// TwinCAT 3 PLC project Untitled1
// ProgramVersion: 3.1.4023.0
// libraries:
//   Tc2_SerialCom, * (Beckhoff Automation GmbH)
//   Tc2_Standard, * (Beckhoff Automation GmbH)
//   Tc2_System, * (Beckhoff Automation GmbH)
//   Tc2_Utilities, * (Beckhoff Automation GmbH)
//   Tc3_Database, * (Beckhoff Automation GmbH)
//   Tc3_IotBase, * (Beckhoff Automation GmbH)
//   Tc3_Module, * (Beckhoff Automation GmbH)
// project tree:
//   DUTs/ ST_SelectStructData.TcDUT, ST_SelectStructIMU.TcDUT (not stored)
//   GVLs/ GVL.TcGVL (not stored)
//   / PlcTask_Background.TcTTO (not stored), PlcTask_Buffer.TcTTO (not stored), PlcTask_Send.TcTTO, PlcTask_Read.TcTTO (not stored), PlcTask_Vacuum.TcTTO
//   POUs/ Background_FatigueCam.TcPOU (not stored), Background_GPS.TcPOU, Background_IMU.TcPOU (not stored), Background_Time.TcPOU, Buffer_Data.TcPOU (not stored), Buffer_IMU.TcPOU, FB_FatigueCam_Receive.TcPOU, Get_Data.TcPOU (not stored), Get_IMU.TcPOU, Main_Background.TcPOU (not stored), Main_Read.TcPOU (not stored), Main_Vacuum.TcPOU, Read_IMU.TcPOU (not stored), Read_Pressure.TcPOU, Read_Payload.TcPOU, Main_Buffer.TcPOU (not stored), Main_Send.TcPOU, Read_FatigueCam.TcPOU (not stored), Read_GPS.TcPOU, Read_ID.TcPOU, Save_Data.TcPOU (not stored), Save_IMU.TcPOU (not stored), Send.TcPOU, Send_IMU.TcPOU, Vacuum_Buffer_Data.TcPOU, Vacuum_Buffer_Data_2.TcPOU, Vacuum_Buffer_IMU.TcPOU, Vacuum_Buffer_IMU_2.TcPOU, Vacuum_Data.TcPOU (not stored), Vacuum_IMU.TcPOU (not stored)

CONFIGURATION Untitled1
    RESOURCE PLC ON TwinCAT3
        TASK PlcTask_Send(INTERVAL := T#4332.9us, PRIORITY := 21);
        TASK PlcTask_Vacuum(INTERVAL := T#333.3us, PRIORITY := 16);
        PROGRAM Main_Send WITH PlcTask_Send : Main_Send;
        PROGRAM Main_Vacuum WITH PlcTask_Vacuum : Main_Vacuum;
    END_RESOURCE
END_CONFIGURATION

// ---- DUTs/ST_SelectStructData.TcDUT
TYPE ST_SelectStructData :
STRUCT
	datetime: STRING(255);
	trailer_id_lead: LINT;
	trailer_id_rear: LINT;
	latitude: REAL;
	longitude: REAL;
	speed: REAL;
	overspeed: LINT;
	payload_lead: REAL;
	payload_rear: REAL;
	overload_lead: LINT;
	overload_rear: LINT;
	pressure_lead: REAL;
	pressure_rear: REAL;
	overpressure_lead: LINT;
	overpressure_rear: LINT;
	event_code: LINT;
END_STRUCT
END_TYPE

// ---- POUs/Main_Send.TcPOU
PROGRAM Main_Send
VAR	
	Done		: BOOL;
	New_Data	: BOOL;
	New_IMU		: BOOL;
	Sent		: BOOL;
	Saved		: BOOL;
	Sent_Data	: BOOL;
	Sent_IMU	: BOOL;
	Saved_Data	: BOOL;
	Saved_IMU	: BOOL;
	
	nState		: INT;

END_VAR

(* get data from database *)
Get_Data();
Get_IMU();

New_Data := Get_Data.Done;
New_IMU := Get_IMU.Done;
 
IF New_Data AND New_IMU THEN
	IF NOT Sent THEN
		(* send data to aws iot core *)
		Send();
		
		IF Send.Published_Data AND Send.Published_IMU THEN
			Sent	:= TRUE;
		END_IF	
		
	ELSE
		IF Save_Data.Done AND Save_IMU.Done THEN
			Saved := TRUE;
		END_IF	
		
	END_IF
	
ELSE
	Sent	:= FALSE;
	Saved 	:= FALSE;
	
END_IF

Save_Data();	
Save_IMU();

END_PROGRAM

// ---- POUs/Get_IMU.TcPOU
PROGRAM Get_IMU
VAR
	fbSqlDatabase	: FB_SQLDatabaseEvt(sNetID := '', tTimeout := T#1000S);
	fbSqlCommand	: FB_SQLCommandEvt(sNetID := '', tTimeout := T#1000S);
	fbSqlCommand2	: FB_SQLCommandEvt(sNetID := '', tTimeout := T#1000S);
	fbSqlResult		: FB_SQLResultEvt(sNetID:='', tTimeout   := T#1000S); 
    aReadStruct		: ARRAY[1..2500] OF ST_SelectStructIMU;
	nState			: INT;
	sCmd			: STRING(20000);
	sCmd2			: STRING(20000);
	val1			: INT;
	val2			: INT;
	exec			: BOOL;
	diff			: BOOL;
	rel				: BOOL;
	exec2			: BOOL;
	diff2			: BOOL;	
	rel2			: BOOL;
	exec3			: BOOL;
	diff3			: BOOL;	
	rel3			: BOOL;
	
	count			: ULINT;
	Data_Length		: ULINT;
	datetime		: STRING;
	Done			: BOOL;
	Deleted			: BOOL := TRUE;
	i 				: ULINT;
	
	TimeStr			: ARRAY[1..2500] OF STRING;	
	Trailer_ID_Lead	: ARRAY[1..2500] OF STRING;
	Trailer_ID_Rear	: ARRAY[1..2500] OF STRING;
	Pitch_Lead		: ARRAY[1..2500] OF STRING;
	Roll_Lead		: ARRAY[1..2500] OF STRING;
	AccX_Lead		: ARRAY[1..2500] OF STRING;
	AccY_Lead		: ARRAY[1..2500] OF STRING;
	AccZ_Lead		: ARRAY[1..2500] OF STRING;
	Pitch_Rear		: ARRAY[1..2500] OF STRING;
	Roll_Rear		: ARRAY[1..2500] OF STRING;
	AccX_Rear		: ARRAY[1..2500] OF STRING;
	AccY_Rear		: ARRAY[1..2500] OF STRING;
	AccZ_Rear		: ARRAY[1..2500] OF STRING;
	
	Dbid			: UDINT;
	Switch			: BOOL;
	Pragma_Done		: BOOL;
	bDisconnect		: BOOL;
	
END_VAR

(* get new data only if prev data sent to aws & saved to localdb *)
IF Main_Send.Saved THEN
	Done	:= FALSE;
	Deleted	:= FALSE;
	IF fbSqlDatabase.bConnected THEN
		nState 	:= 1;
	ELSE
		nState 	:= 0;
	END_IF
END_IF

IF Switch THEN
	IF Buffer_IMU.Dbid = Dbid AND Buffer_IMU.fbSqlDatabase.bConnected THEN
		Switch := FALSE;
	END_IF
	
ELSIF Buffer_IMU.Initialized AND Buffer_IMU.fbSqlDatabase.bConnected THEN
	
	CASE nState OF
		
		0:
			//choose db opposite of buffer
			IF Buffer_IMU.Dbid = 2 THEN
				Dbid := 5;
			ELSE
				Dbid := 2;
			END_IF
			
			IF fbSqlDatabase.Connect(Dbid) THEN
				IF fbSqlDatabase.bError THEN
					nState := 255;
				ELSE
					nState := nState + 1;
				END_IF
			END_IF
			
		1:
			IF fbSqlDatabase.CreateCmd(ADR(fbSqlCommand)) THEN
				IF fbSqlDatabase.bError THEN
					nState := 255; 
				ELSE
					nState := nState+1; 
				END_IF
			END_IF
			
		2:	(* execute pragmas *)
			IF NOT Pragma_Done THEN
				sCmd	:= 'PRAGMA journal_mode = WAL; PRAGMA synchronous = NORMAL; PRAGMA temp_store = MEMORY; PRAGMA mmap_size = 30000000000; PRAGMA page_size = 32768; PRAGMA locking_mode = EXCLUSIVE;';
			
				IF fbSQLCommand.Execute(ADR(sCmd), SIZEOF(sCmd)) THEN
					IF fbSQLCommand.bError THEN
						nState := 255; 
					ELSE
						nState 		:= nState+1; 
						Pragma_Done := TRUE;
					END_IF
				END_IF
			
			ELSE
				nState 		:= nState+1;
			END_IF
		
		3:	
			IF Deleted THEN
				nState := nState+1;
			ELSE
				(* delete saved data from buffer *)
				sCmd2	:= 'DELETE FROM buffer_imu WHERE datetime IN (SELECT datetime FROM buffer_imu ORDER BY datetime ASC LIMIT ';
				sCmd2	:= CONCAT(sCmd2, ULINT_TO_STRING(Data_Length));
				sCmd2	:= CONCAT(sCmd2, ');');
				
				IF fbSQLCommand.Execute(ADR(sCmd2), SIZEOF(sCmd2)) THEN
					IF fbSQLCommand.bError THEN
						nState := 255; 
					ELSE
						nState := nState+1; 
						Deleted := TRUE;
					END_IF
				END_IF
			END_IF
			
		4:	
			(* count no of records in buffer *)
			sCmd2 := 'SELECT COUNT(*) FROM `buffer_imu`';
			
			IF fbSQLCommand.ExecuteDataReturn(ADR(sCmd2), SIZEOF(sCmd2), ADR(fbSqlResult)) THEN
				IF fbSQLCommand.bError THEN
					nState := 255; 
				ELSE
					nState := nState+1; 
				END_IF
			END_IF
			
		5:	
			IF fbSqlResult.Read(0, 1, ADR(count), SIZEOF(count), TRUE, TRUE) THEN
				IF fbSqlResult.bError THEN
					nState := 255; 
				ELSE
					nState := nState+1; 
				END_IF
			END_IF
			
		6:
			IF fbSqlResult.Release() THEN
				IF fbSqlResult.bError THEN
					nState := 255;
				ELSE
					nState := nState + 1;
				END_IF
				
			END_IF
			
		7:
			(* determine no of records to select *)
			IF count = 0 THEN
				Data_Length := 0;
				nState := 13;
			
			ELSIF count < 1000 THEN
				Data_Length := count;
				nState := nState+1;
			
			ELSE
				Data_Length := 1000;
				nState := nState+1;
			
			END_IF
			
		8:	
			(* get records from buffer *)
			sCmd2 := 'SELECT * FROM `buffer_imu` ORDER BY datetime ASC LIMIT ';
			sCmd2 := CONCAT(sCmd2, ULINT_TO_STRING(Data_Length));
			
			IF fbSQLCommand.ExecuteDataReturn(ADR(sCmd2), SIZEOF(sCmd2), ADR(fbSqlResult)) THEN
				IF fbSQLCommand.bError THEN
					nState := 255; 
				ELSE
					nState := nState+1; 
				END_IF
			END_IF
			
		9:
			IF fbSqlResult.Read(0, ULINT_TO_UDINT(Data_Length), ADR(aReadStruct), SIZEOF(aReadStruct), TRUE, TRUE) THEN
				IF fbSqlResult.bError THEN
					nState := 255; 
				ELSE
					nState := nState+1; 
				END_IF
			END_IF
			
		10:
			IF fbSqlResult.Release() THEN
				IF fbSqlResult.bError THEN
					nState := 255;
				ELSE
					nState := nState+1;
				END_IF
			END_IF
		
		11:
			(* parse query result *)
			FOR i:=1 TO Data_Length BY 1 DO
				TimeStr[i]			:= aReadStruct[i].datetime;
				
				Trailer_ID_Lead[i]			:= LINT_TO_STRING(aReadStruct[i].trailer_id_lead);
				Trailer_ID_Rear[i]			:= LINT_TO_STRING(aReadStruct[i].trailer_id_rear);
				//RoadSec[i]				:= UINT_TO_STRING(aReadStruct[i].RoadSec);
				Pitch_Lead[i]				:= REAL_TO_STRING(aReadStruct[i].pitch_lead);
				Roll_Lead[i]				:= REAL_TO_STRING(aReadStruct[i].roll_lead);
				AccX_Lead[i]				:= REAL_TO_STRING(aReadStruct[i].ax_lead);
				AccY_Lead[i]				:= REAL_TO_STRING(aReadStruct[i].ay_lead);
				AccZ_Lead[i]				:= REAL_TO_STRING(aReadStruct[i].az_lead);
				Pitch_Rear[i]				:= REAL_TO_STRING(aReadStruct[i].pitch_rear);
				Roll_Rear[i]				:= REAL_TO_STRING(aReadStruct[i].roll_rear);
				AccX_Rear[i]				:= REAL_TO_STRING(aReadStruct[i].ax_rear);
				AccY_Rear[i]				:= REAL_TO_STRING(aReadStruct[i].ay_rear);
				AccZ_Rear[i]				:= REAL_TO_STRING(aReadStruct[i].az_rear);
				
			END_FOR
			
			nState	:= nState + 1;
			
		12:
			Done	:= TRUE;
			
		13:	(* execute pragma optimize *)
			sCmd	:= 'PRAGMA optimize;';
			
			IF fbSQLCommand.Execute(ADR(sCmd), SIZEOF(sCmd)) THEN
				IF fbSQLCommand.bError THEN
					nState := 255; 
				ELSE
					nState := nState+1; 
				END_IF
			END_IF
			
		14:
			//disconnect from db
			IF bDisconnect := fbSqlDatabase.Disconnect() THEN
				IF fbSqlDatabase.bError THEN
					nState := 255;
				ELSE
					nState 		:= 0;
					Switch 		:= TRUE;
					Pragma_Done	:= FALSE;
				END_IF
			END_IF			
		
		255:
			nState	:= 0;	
			
	END_CASE
	
END_IF

END_PROGRAM

// ---- POUs/Buffer_IMU.TcPOU
PROGRAM Buffer_IMU
VAR
	pSec		: WORD;
	diff		: BOOL;
	
	TimeStr		: ARRAY [1..50] OF STRING;
	//Millis		: ARRAY [1..50] OF STRING;
	Trailer_ID_Lead	: ARRAY [1..50] OF STRING;
	//RoadSec		: ARRAY [1..50] OF STRING;
	Pitch_Lead		: ARRAY [1..50] OF STRING;
	Roll_Lead		: ARRAY [1..50] OF STRING;
	AccX_Lead		: ARRAY [1..50] OF STRING;
	AccY_Lead		: ARRAY [1..50] OF STRING;
	AccZ_Lead		: ARRAY [1..50] OF STRING;
	
	Trailer_ID_Rear	: ARRAY [1..50] OF STRING;
	//RoadSec		: ARRAY [1..50] OF STRING;
	Pitch_Rear		: ARRAY [1..50] OF STRING;
	Roll_Rear		: ARRAY [1..50] OF STRING;
	AccX_Rear		: ARRAY [1..50] OF STRING;
	AccY_Rear		: ARRAY [1..50] OF STRING;
	AccZ_Rear		: ARRAY [1..50] OF STRING;
	
	fbSqlDatabase	: FB_SQLDatabaseEvt(sNetID := '', tTimeout := T#1000S);
	fbSqlCommand	: FB_SQLCommandEvt(sNetID := '', tTimeout := T#1000S);
	fbSqlResult		: FB_SQLResultEvt(sNetID:='', tTimeout   := T#1000S); 
	sCmd			: STRING(500000);
	sCmd2			: STRING(500000);
	nState			: INT;
	nState_Switch	: INT;
	
	aReadStruct		: ST_SelectStructIMU;
	aReadStruct_2	: ST_SelectStructIMU;
	Timestamp		: DT;
	Timestamp_2		: DT; 
	
	Initialized		: BOOL := FALSE;
	Done			: BOOL;
	i				: INT;
	Pragma_Done		: BOOL;
	Counter			: ULINT;
	
	Dbid			: UDINT;
	
	bDisconnect		: BOOL;
END_VAR

(* convert to strings *)
//PrimeMover_ID		:= Read_ID.PrimeMover_ID;
TimeStr				:= Read_IMU.TimeStr;
//Millis			:= Read_IMU.Millis;
Trailer_ID_Lead		:= Read_IMU.Trailer_ID_Lead;
Pitch_Lead			:= Read_IMU.Pitch_Lead;
Roll_Lead			:= Read_IMU.Roll_Lead;
AccX_Lead			:= Read_IMU.AccX_Lead;
AccY_Lead			:= Read_IMU.AccY_Lead;
AccZ_Lead			:= Read_IMU.AccZ_Lead;

Trailer_ID_Rear		:= Read_IMU.Trailer_ID_Rear;
Pitch_Rear			:= Read_IMU.Pitch_Rear;
Roll_Rear			:= Read_IMU.Roll_Rear;
AccX_Rear			:= Read_IMU.AccX_Rear;
AccY_Rear			:= Read_IMU.AccY_Rear;
AccZ_Rear			:= Read_IMU.AccZ_Rear;

IF NOT Initialized THEN
	
	//initialization (choose which database for buffer)
	CASE nState OF
				
		0:
			(* connect to buffer_imu *)	
			IF Vacuum_Buffer_IMU.Vacuumed THEN
				
				Dbid := 2;		
				IF fbSqlDatabase.Connect(Dbid) THEN
					IF fbSqlDatabase.bError THEN
						nState := 255; 
					ELSE
						nState := nState+1;
					END_IF
				END_IF
				
			END_IF
			
			
		1:
			IF fbSqlDatabase.CreateCmd(ADR(fbSqlCommand)) THEN
				IF fbSqlDatabase.bError THEN
					nState := 255; 
				ELSE
					nState := nState+1; 
				END_IF
			END_IF
			
		2:	(* execute pragmas *)
			sCmd	:= 'PRAGMA journal_mode = WAL; PRAGMA synchronous = NORMAL; PRAGMA temp_store = MEMORY; PRAGMA mmap_size = 30000000000; PRAGMA page_size = 32768; PRAGMA locking_mode = EXCLUSIVE;';
			
			IF fbSQLCommand.Execute(ADR(sCmd), SIZEOF(sCmd)) THEN
				IF fbSQLCommand.bError THEN
					nState := 255; 
				ELSE
					nState := nState+1; 
				END_IF
			END_IF
			
		3:
			(* select oldest data from buffer_imu *)
			sCmd	:= 'SELECT * FROM `buffer_imu` ORDER BY datetime ASC LIMIT 1';
			
			IF fbSQLCommand.ExecuteDataReturn(ADR(sCmd), SIZEOF(sCmd), ADR(fbSqlResult)) THEN
				IF fbSQLCommand.bError THEN
					nState := 255; 
				ELSE
					nState := nState+1; 
				END_IF
			END_IF
			
		4:
			IF fbSqlResult.Read(0, 1, ADR(aReadStruct), SIZEOF(aReadStruct), TRUE, TRUE) THEN
				IF fbSqlResult.bError THEN
					nState := 255; 
				ELSE
					nState := nState+1; 
				END_IF
			END_IF
			
		5:
			IF fbSqlResult.Release() THEN
				IF fbSqlResult.bError THEN
					nState := 255;
				ELSE
					nState := nState+1;
				END_IF
			END_IF
			
		6:	(* execute pragma optimize *)
			sCmd	:= 'PRAGMA optimize;';
			
			IF fbSQLCommand.Execute(ADR(sCmd), SIZEOF(sCmd)) THEN
				IF fbSQLCommand.bError THEN
					nState := 255; 
				ELSE
					nState := nState+1; 
				END_IF
			END_IF
			
		7:
			(* disconnect from buffer_imu *)
			IF fbSqlDatabase.Disconnect() THEN
				IF fbSqlDatabase.bError THEN
					nState := 255;
				ELSE
					nState := nState+1;
				END_IF
			END_IF
			
		8:	
			(* connect to buffer_imu_2 *)
			IF Vacuum_Buffer_IMU_2.Vacuumed THEN
				
				Dbid := 5;	
				IF fbSqlDatabase.Connect(Dbid) THEN
					IF fbSqlDatabase.bError THEN
						nState := 255; 
					ELSE
						nState := nState+1;
					END_IF
				END_IF
				
			END_IF	
			
		9:
			IF fbSqlDatabase.CreateCmd(ADR(fbSqlCommand)) THEN
				IF fbSqlDatabase.bError THEN
					nState := 255; 
				ELSE
					nState := nState+1; 
				END_IF
			END_IF
			
		10:	(* execute pragmas *)
			sCmd	:= 'PRAGMA journal_mode = WAL; PRAGMA synchronous = NORMAL; PRAGMA temp_store = MEMORY; PRAGMA mmap_size = 30000000000; PRAGMA page_size = 32768; PRAGMA locking_mode = EXCLUSIVE;';
			
			IF fbSQLCommand.Execute(ADR(sCmd), SIZEOF(sCmd)) THEN
				IF fbSQLCommand.bError THEN
					nState := 255; 
				ELSE
					nState := nState+1; 
				END_IF
			END_IF
			
		11:
			(* select oldest data from buffer_imu *)
			sCmd	:= 'SELECT * FROM `buffer_imu` ORDER BY datetime ASC LIMIT 1';
			
			IF fbSQLCommand.ExecuteDataReturn(ADR(sCmd), SIZEOF(sCmd), ADR(fbSqlResult)) THEN
				IF fbSQLCommand.bError THEN
					nState := 255; 
				ELSE
					nState := nState+1; 
				END_IF
			END_IF
			
		12:
			IF fbSqlResult.Read(0, 1, ADR(aReadStruct_2), SIZEOF(aReadStruct_2), TRUE, TRUE) THEN
				IF fbSqlResult.bError THEN
					nState := 255; 
				ELSE
					nState := nState+1; 
				END_IF
			END_IF
			
		13:
			IF fbSqlResult.Release() THEN
				IF fbSqlResult.bError THEN
					nState := 255;
				ELSE
					nState := nState+1;
				END_IF
			END_IF
			
		14:	(* execute pragma optimize *)
			sCmd	:= 'PRAGMA optimize;';
			
			IF fbSQLCommand.Execute(ADR(sCmd), SIZEOF(sCmd)) THEN
				IF fbSQLCommand.bError THEN
					nState := 255; 
				ELSE
					nState := nState+1; 
				END_IF
			END_IF
			
		15:
			(* disconnect from buffer_imu_2 *)
			IF bDisconnect := fbSqlDatabase.Disconnect() THEN
				IF fbSqlDatabase.bError THEN
					nState := 255;
				ELSE
					nState := nState+1;
				END_IF
			END_IF
			
		16:
			// compare oldest data
			aReadStruct.datetime 	:= REPLACE(aReadStruct.datetime, '-', 1, 11);
			aReadStruct_2.datetime 	:= REPLACE(aReadStruct_2.datetime, '-', 1, 11);
			
			Timestamp	:= SYSTEMTIME_TO_DT(STRING_TO_SYSTEMTIME(aReadStruct.datetime));
			Timestamp_2	:= SYSTEMTIME_TO_DT(STRING_TO_SYSTEMTIME(aReadStruct_2.datetime));

			IF Timestamp = DT#1970-1-1-00:00:00 THEN
				Dbid := 2;
			ELSIF Timestamp_2 = DT#1970-1-1-00:00:00 THEN
				Dbid := 5;
			ELSIF Timestamp > Timestamp_2 THEN
				Dbid := 2;
			ELSE
				Dbid := 5;
			END_IF
			
			Initialized := TRUE;
			nState		:= 0;
			
		255:
			nState := 0;
			
	END_CASE

ELSE	
	
	(* save data to buffer every second *)
	IF diff:= Background_Time.cSec <> pSec THEN
		
		//database switching
		IF Get_IMU.Switch AND Counter >= 250 THEN
			
			CASE nState_Switch OF
				
				0:	(* execute pragma optimize *)
					sCmd	:= 'PRAGMA optimize;';
					
					IF fbSQLCommand.Execute(ADR(sCmd), SIZEOF(sCmd)) THEN
						IF fbSQLCommand.bError THEN
							nState_Switch := 255; 
						ELSE
							nState_Switch := nState_Switch+1; 
						END_IF
					END_IF
				
				1:
					IF fbSqlDatabase.bConnected THEN
						fbSqlDatabase.Disconnect();
					ELSE
						IF Dbid = 2 THEN
							Dbid := 5;
						ELSE
							Dbid := 2;
						END_IF
						Counter			:= 0;
						nState_Switch 	:= 0;
						Pragma_Done		:= FALSE;
					END_IF
					
				255:
					nState_Switch := 0;
					
			END_CASE
		
		ELSE
			
			IF Done THEN
				Done	:= FALSE;
				IF fbSqlDatabase.bConnected THEN
					nState 	:= 1;
				ELSE
					nState 	:= 0;
				END_IF	
			END_IF
			
			CASE nState OF	
				0:	
					IF fbSqlDatabase.Connect(Dbid) THEN
						IF fbSqlDatabase.bError THEN
							nState := 255;
						ELSE
							nState := nState + 1; 
						END_IF
					END_IF
				
				1:
					IF fbSqlDatabase.CreateCmd(ADR(fbSqlCommand)) THEN
						IF fbSqlDatabase.bError THEN
							nState := 255; 
						ELSE
							nState := nState+1; 
						END_IF
					END_IF
					
				2:	(* execute pragmas *)
					IF NOT Pragma_Done THEN
						sCmd	:= 'PRAGMA journal_mode = WAL; PRAGMA synchronous = NORMAL; PRAGMA temp_store = MEMORY; PRAGMA mmap_size = 30000000000; PRAGMA page_size = 32768; PRAGMA locking_mode = EXCLUSIVE;';
					
						IF fbSQLCommand.Execute(ADR(sCmd), SIZEOF(sCmd)) THEN
							IF fbSQLCommand.bError THEN
								nState := 255; 
							ELSE
								nState 		:= nState+1; 
								Pragma_Done := TRUE;
							END_IF
						END_IF
					
					ELSE
						nState 		:= nState+1;
 
					END_IF
					
				3:	
					(* build query *)	
					sCmd:= 'INSERT INTO buffer_imu (datetime,trailer_id_lead,trailer_id_rear,pitch_lead,roll_lead,ax_lead,ay_lead,az_lead,pitch_rear,roll_rear,ax_rear,ay_rear,az_rear) VALUES ';
					
					FOR i := 1 TO 50 BY 1 DO
						sCmd2:= CONCAT('($'', TimeStr[i]);
						sCmd2:= CONCAT(sCmd2, '$',');
						sCmd2:= CONCAT(sCmd2, Trailer_ID_Lead[i]);
						sCmd2:= CONCAT(sCmd2, ',');
						sCmd2:= CONCAT(sCmd2, Trailer_ID_Rear[i]);
						sCmd2:= CONCAT(sCmd2, ',');
						sCmd2:= CONCAT(sCmd2, Pitch_Lead[i]);
						sCmd2:= CONCAT(sCmd2, ',');
						sCmd2:= CONCAT(sCmd2, Roll_Lead[i]);
						sCmd2:= CONCAT(sCmd2, ',');
						sCmd2:= CONCAT(sCmd2, AccX_Lead[i]);
						sCmd2:= CONCAT(sCmd2, ',');
						sCmd2:= CONCAT(sCmd2, AccY_Lead[i]);
						sCmd2:= CONCAT(sCmd2, ',');
						sCmd2:= CONCAT(sCmd2, AccZ_Lead[i]);
						sCmd2:= CONCAT(sCmd2, ',');
						sCmd2:= CONCAT(sCmd2, Pitch_Rear[i]);
						sCmd2:= CONCAT(sCmd2, ',');
						sCmd2:= CONCAT(sCmd2, Roll_Rear[i]);
						sCmd2:= CONCAT(sCmd2, ',');
						sCmd2:= CONCAT(sCmd2, AccX_Rear[i]);
						sCmd2:= CONCAT(sCmd2, ',');
						sCmd2:= CONCAT(sCmd2, AccY_Rear[i]);
						sCmd2:= CONCAT(sCmd2, ',');
						sCmd2:= CONCAT(sCmd2, AccZ_Rear[i]);
						
						IF i = 50 THEN
							sCmd2:= CONCAT(sCmd2, ')');
						ELSE	
							sCmd2:= CONCAT(sCmd2, '),');
						END_IF
						
						CONCAT2(ADR(sCmd), ADR(sCmd2), ADR(sCmd), SIZEOF(sCmd));
					END_FOR
					
					
					IF fbSQLCommand.Execute(ADR(sCmd), SIZEOF(sCmd)) THEN
						IF fbSQLCommand.bError THEN
							nState := 255; 
						ELSE
							nState := nState+1; 
							pSec := Background_Time.cSec;
							
						END_IF
					END_IF
					
				4: 
					Counter := Counter + 50;
					Done	:= TRUE;
						
				255:
					nState := 0;
					
			END_CASE	
			
		END_IF
	END_IF
END_IF

END_PROGRAM

// ---- POUs/Vacuum_Buffer_IMU.TcPOU
PROGRAM Vacuum_Buffer_IMU
VAR
	fbSqlDatabase	: FB_SQLDatabaseEvt(sNetID := '', tTimeout := T#1000S);
	fbSqlCommand	: FB_SQLCommandEvt(sNetID := '', tTimeout := T#1000S);
	fbSqlResult		: FB_SQLResultEvt(sNetID :='', tTimeout   := T#1000S); 
	nState			: INT;
	sCmd			: STRING(500000);
	Vacuumed		: BOOL;
END_VAR

CASE nState OF
				
		0:
			(* connect to buffer_imu *)		
			IF fbSqlDatabase.Connect(2) THEN
				IF fbSqlDatabase.bError THEN
					nState := 255; 
				ELSE
					IF fbSqlDatabase.bConnected THEN
						nState := nState+1;
					END_IF 
				END_IF
			END_IF
			
		1:
			IF fbSqlDatabase.CreateCmd(ADR(fbSqlCommand)) THEN
				IF fbSqlDatabase.bError THEN
					nState := 255; 
				ELSE
					nState := nState+1; 
				END_IF
			END_IF
			
		2:	(* execute pragmas *)
			sCmd	:= 'PRAGMA journal_mode = WAL; PRAGMA synchronous = NORMAL; PRAGMA temp_store = MEMORY; PRAGMA mmap_size = 30000000000; PRAGMA page_size = 32768; PRAGMA locking_mode = EXCLUSIVE;';
			
			IF fbSQLCommand.Execute(ADR(sCmd), SIZEOF(sCmd)) THEN
				IF fbSQLCommand.bError THEN
					nState := 255; 
				ELSE
					nState := nState+1; 
				END_IF
			END_IF
		
		3:	
			IF NOT Vacuumed THEN
				(* build query *)	
				sCmd	:= 'VACUUM';
				
				IF fbSQLCommand.Execute(ADR(sCmd), SIZEOF(sCmd)) THEN
					IF fbSQLCommand.bError THEN
						nState := 255; 
					ELSE
						nState 		:= nState+1; 
					END_IF
				END_IF
				
			ELSE 
				nState := nState+1;
			END_IF
			
		4:	(* execute pragma optimize *)
			sCmd	:= 'PRAGMA optimize;';
			
			IF fbSQLCommand.Execute(ADR(sCmd), SIZEOF(sCmd)) THEN
				IF fbSQLCommand.bError THEN
					nState := 255; 
				ELSE
					nState := nState+1; 
				END_IF
			END_IF
		
		5:
			IF fbSqlDatabase.Disconnect() THEN
				IF fbSqlDatabase.bError THEN
					nState := 255;
				ELSE
					nState 		:= nState+1;
					Vacuumed 	:= TRUE;
				END_IF
			END_IF
			
		255:
			nState := 0;
	
END_CASE

END_PROGRAM

// ---- POUs/Vacuum_Buffer_IMU_2.TcPOU
PROGRAM Vacuum_Buffer_IMU_2
VAR
	fbSqlDatabase	: FB_SQLDatabaseEvt(sNetID := '', tTimeout := T#1000S);
	fbSqlCommand	: FB_SQLCommandEvt(sNetID := '', tTimeout := T#1000S);
	fbSqlResult		: FB_SQLResultEvt(sNetID :='', tTimeout   := T#1000S); 
	nState			: INT;
	sCmd			: STRING(500000);
	Vacuumed		: BOOL;
END_VAR

CASE nState OF
				
		0:
			(* connect to buffer_imu *)		
			IF fbSqlDatabase.Connect(5) THEN
				IF fbSqlDatabase.bError THEN
					nState := 255; 
				ELSE
					IF fbSqlDatabase.bConnected THEN
						nState := nState+1;
					END_IF 
				END_IF
			END_IF
			
		1:
			IF fbSqlDatabase.CreateCmd(ADR(fbSqlCommand)) THEN
				IF fbSqlDatabase.bError THEN
					nState := 255; 
				ELSE
					nState := nState+1; 
				END_IF
			END_IF
			
		2:	(* execute pragmas *)
			sCmd	:= 'PRAGMA journal_mode = WAL; PRAGMA synchronous = NORMAL; PRAGMA temp_store = MEMORY; PRAGMA mmap_size = 30000000000; PRAGMA page_size = 32768; PRAGMA locking_mode = EXCLUSIVE;';
			
			IF fbSQLCommand.Execute(ADR(sCmd), SIZEOF(sCmd)) THEN
				IF fbSQLCommand.bError THEN
					nState := 255; 
				ELSE
					nState := nState+1; 
				END_IF
			END_IF
		
		3:	
			IF NOT Vacuumed THEN
				(* build query *)	
				sCmd	:= 'VACUUM';
				
				IF fbSQLCommand.Execute(ADR(sCmd), SIZEOF(sCmd)) THEN
					IF fbSQLCommand.bError THEN
						nState := 255; 
					ELSE
						nState 		:= nState+1; 
					END_IF
				END_IF
				
			ELSE 
				nState := nState+1;
			END_IF
			
		4:	(* execute pragma optimize *)
			sCmd	:= 'PRAGMA optimize;';
			
			IF fbSQLCommand.Execute(ADR(sCmd), SIZEOF(sCmd)) THEN
				IF fbSQLCommand.bError THEN
					nState := 255; 
				ELSE
					nState := nState+1; 
				END_IF
			END_IF
		
		5:
			IF fbSqlDatabase.Disconnect() THEN
				IF fbSqlDatabase.bError THEN
					nState := 255;
				ELSE
					nState 		:= nState+1;
					Vacuumed 	:= TRUE;
				END_IF
			END_IF
			
		255:
			nState := 0;
			
END_CASE

END_PROGRAM

// ---- POUs/Background_Time.TcPOU
PROGRAM Background_Time
VAR
	fbTime 		: FB_LocalSystemTime := ( bEnable := TRUE, dwCycle := 1 );
	bValid		: BOOL := FALSE;
	TimeStr		: STRING;
	cSec		: WORD;
	cMil		: WORD;
END_VAR

(* get system time *)
WHILE bValid = FALSE DO
	fbTime(bValid => bValid);	
END_WHILE

fbTime();

TimeStr	:= SYSTEMTIME_TO_STRING(Background_Time.fbTime.systemTime);
cSec	:= fbTime.systemTime.wSecond;
cMil	:= fbTime.systemTime.wMilliseconds;

END_PROGRAM

// ---- POUs/Send.TcPOU
PROGRAM Send
VAR
	fbMqttClient : FB_IotMqttClient;
	bSetParameter : BOOL := TRUE;
	bConnect : BOOL := TRUE;
	
	(* aws certificates *)
	
	(*------------------ actual ----------------*)
	(*
	rootCA		: STRING(255) := 'C:\Users\Administrator\Downloads\AWSCert\AmazonRootCA1.pem';
	thingCert	: STRING(255) := 'C:\Users\Administrator\Downloads\AWSCert\a2ca8bd1ed97a43e38f2bffcdf7ca64a29d3483826fdb03b3eb616af8a5efc9e-certificate.pem.crt';
	privateKey	: STRING(255) := 'C:\Users\Administrator\Downloads\AWSCert\a2ca8bd1ed97a43e38f2bffcdf7ca64a29d3483826fdb03b3eb616af8a5efc9e-private.pem.key';
	*)
	
	rootCA		: STRING(255) := 'C:\Users\Administrator\Downloads\AWSCert\AmazonRootCA1.pem';
	thingCert	: STRING(255) := 'C:\Users\Administrator\Downloads\AWSCert\30ca1f75dd1439c7068842e0254dcd64758e3e884a9c2ab8cf28b27caf6d120f-certificate.pem.crt';
	privateKey	: STRING(255) := 'C:\Users\Administrator\Downloads\AWSCert\30ca1f75dd1439c7068842e0254dcd64758e3e884a9c2ab8cf28b27caf6d120f-private.pem.key';
	
	(* ------------------ test ------------------ *)
	(*
	rootCA		: STRING(255) := 'C:\Users\muhammad.rahman\Downloads\double-sdt-1-certs\AmazonRootCA1.pem';
	thingCert	: STRING(255) := 'C:\Users\muhammad.rahman\Downloads\double-sdt-test-certs\8872c9f9d2c9335079f20c0506a3dd3599fd4d8552622bd2d7f8ae6d1681c64f-certificate.pem.crt';
	privateKey	: STRING(255) := 'C:\Users\muhammad.rahman\Downloads\double-sdt-test-certs\8872c9f9d2c9335079f20c0506a3dd3599fd4d8552622bd2d7f8ae6d1681c64f-private.pem.key';
	*)
	
	(* broker settings *)
	endpoint	: STRING := 'a2o01t3xth0mr1-ats.iot.ap-southeast-1.amazonaws.com';
	port		: UINT := 8883;
	clientID	: STRING := 'double-sdt-2';
	//clientID	: STRING := 'double-sdt-test';
	
	(* published message *)
	sTopicPub 		: STRING(255) := 'iot/smartproduct/mifa/double-sdt/data'; //message topic
	sTopicPub_2 	: STRING(255) := 'iot/smartproduct/mifa/double-sdt/imu'; //message topic
	sPayloadPub 	: STRING(50000000);
	str				: STRING(10000000);
	valSeparator	: STRING := '","';
	comma			: STRING := ',';
	arrayEnd		: STRING := '"]';
	arrayEnd2		: STRING := ']';
	msgEnd			: STRING := '}';
	i				: ULINT;
	
	(* topic subscription *)
	bSubscribed : BOOL;
	sTopicSub 	: STRING(255) := 'iot/smartproduct/mifa/double-sdt/data';
	sTopicSub_2	: STRING(255) := 'iot/smartproduct/mifa/double-sdt/imu';
	
	(* received message *)	
	{attribute 'TcEncoding':='UTF-8'}
	sTopicRcv : STRING(255);
	{attribute 'TcEncoding':='UTF-8'}
	sPayloadRcv : STRING(255);
	
	fbMessageQueue : FB_IotMqttMessageQueue;
	fbMessage : FB_IotMqttMessage;
	
	hrErrorOccurred : HRESULT; // contains the latest occurred error
	
	Published_Data		: BOOL;
	Publish_Data		: BOOL;
	Published_IMU		: BOOL;
	Publish_IMU			: BOOL;
END_VAR

IF bSetParameter THEN
	bSetParameter := FALSE;
	
	(* TLS settings for AWS IoT connection *)
	fbMqttClient.stTLS.sCA 		:= rootCA; //root CA
    fbMqttClient.stTLS.sCert 	:= thingCert; //certificate of thing
    fbMqttClient.stTLS.sKeyFile := privateKey; //private key of thing
	
	(* Broker settings für AWS IoT *)
	fbMqttClient.sHostName:= endpoint; //broker endpoint
	fbMqttClient.nHostPort:= port; //default mqtt tls port
	fbMqttClient.sClientId:= clientID; //client id
	fbMqttClient.sTopicPrefix:= ''; 
	
	fbMqttClient.ipMessageQueue := fbMessageQueue;
END_IF

(* connect to mqtt broker *)
fbMqttClient.Execute(bConnect); 
IF fbMqttClient.bError THEN
	// add your error logging here
	hrErrorOccurred := fbMqttClient.hrErrorCode;
END_IF

(* send data *)
IF Main_Send.New_Data THEN
	Publish_Data		:= FALSE;
	Published_Data	 	:= FALSE;	
	
	IF fbMqttClient.bConnected THEN	
		IF NOT bSubscribed THEN
			bSubscribed := fbMqttClient.Subscribe(sTopic:=sTopicSub, eQoS:=TcIotMqttQos.AtMostOnceDelivery); //subscribe to topic
			IF fbMqttClient.bError THEN
				// add your error logging here
				hrErrorOccurred := fbMqttClient.hrErrorCode;
			END_IF
		END_IF
		
		(* build message payload *)
		sPayloadPub := CONCAT('{"primemover_id":', Read_ID.PrimeMover_ID);
		
		(* lead trailer id string *)
		str	:= ',"trailer_id_lead":[';
		FOR i:=1 TO Get_Data.Data_Length BY 1 DO
			CONCAT2(ADR(str), ADR(Get_Data.Trailer_ID_Lead[i]), ADR(str), SIZEOF(str)); 
			
			IF i <> Get_Data.Data_Length THEN
				CONCAT2(ADR(str), ADR(comma), ADR(str), SIZEOF(str));
			ELSE
				CONCAT2(ADR(str), ADR(arrayEnd2), ADR(str), SIZEOF(str));
			END_IF
			
		END_FOR
		
		CONCAT2(ADR(sPayloadPub), ADR(str), ADR(sPayloadPub), SIZEOF(sPayloadPub));
		
		(* rear trailer id string *)
		str	:= ',"trailer_id_rear":[';
		FOR i:=1 TO Get_Data.Data_Length BY 1 DO
			CONCAT2(ADR(str), ADR(Get_Data.Trailer_ID_Rear[i]), ADR(str), SIZEOF(str)); 
			
			IF i <> Get_Data.Data_Length THEN
				CONCAT2(ADR(str), ADR(comma), ADR(str), SIZEOF(str));
			ELSE
				CONCAT2(ADR(str), ADR(arrayEnd2), ADR(str), SIZEOF(str));
			END_IF
			
		END_FOR
		
		CONCAT2(ADR(sPayloadPub), ADR(str), ADR(sPayloadPub), SIZEOF(sPayloadPub));
		
		(* date time string *)
		str	:= ',"datetime":["';
		FOR i:=1 TO Get_Data.Data_Length BY 1 DO
			CONCAT2(ADR(str), ADR(Get_Data.TimeStr[i]), ADR(str), SIZEOF(str)); 
			
			IF i <> Get_Data.Data_Length THEN
				CONCAT2(ADR(str), ADR(valSeparator), ADR(str), SIZEOF(str));
			ELSE
				CONCAT2(ADR(str), ADR(arrayEnd), ADR(str), SIZEOF(str));
			END_IF
			
		END_FOR
		
		CONCAT2(ADR(sPayloadPub), ADR(str), ADR(sPayloadPub), SIZEOF(sPayloadPub));
		
		(* latitude string *)
		str	:= ',"latitude":[';
		FOR i:=1 TO Get_Data.Data_Length BY 1 DO
			CONCAT2(ADR(str), ADR(Get_Data.Lat[i]), ADR(str), SIZEOF(str)); 
			
			IF i <> Get_Data.Data_Length THEN
				CONCAT2(ADR(str), ADR(comma), ADR(str), SIZEOF(str));
			ELSE
				CONCAT2(ADR(str), ADR(arrayEnd2), ADR(str), SIZEOF(str));
			END_IF
			
		END_FOR
		
		CONCAT2(ADR(sPayloadPub), ADR(str), ADR(sPayloadPub), SIZEOF(sPayloadPub));
		
		(* longitude string *)
		str	:= ',"longitude":[';
		FOR i:=1 TO Get_Data.Data_Length BY 1 DO
			CONCAT2(ADR(str), ADR(Get_Data.Lon[i]), ADR(str), SIZEOF(str)); 
			
			IF i <> Get_Data.Data_Length THEN
				CONCAT2(ADR(str), ADR(comma), ADR(str), SIZEOF(str));
			ELSE
				CONCAT2(ADR(str), ADR(arrayEnd2), ADR(str), SIZEOF(str));
			END_IF
			
		END_FOR
		
		CONCAT2(ADR(sPayloadPub), ADR(str), ADR(sPayloadPub), SIZEOF(sPayloadPub));
		
		(* speed string *)
		str	:= ',"speed":[';
		FOR i:=1 TO Get_Data.Data_Length BY 1 DO
			CONCAT2(ADR(str), ADR(Get_Data.Speed[i]), ADR(str), SIZEOF(str)); 
			
			IF i <> Get_Data.Data_Length THEN
				CONCAT2(ADR(str), ADR(comma), ADR(str), SIZEOF(str));
			ELSE
				CONCAT2(ADR(str), ADR(arrayEnd2), ADR(str), SIZEOF(str));
			END_IF
			
		END_FOR
		
		CONCAT2(ADR(sPayloadPub), ADR(str), ADR(sPayloadPub), SIZEOF(sPayloadPub));
		
		(* overspeed string *)
		str	:= ',"overspeed":[';
		FOR i:=1 TO Get_Data.Data_Length BY 1 DO
			CONCAT2(ADR(str), ADR(Get_Data.Overspeed[i]), ADR(str), SIZEOF(str)); 
			
			IF i <> Get_Data.Data_Length THEN
				CONCAT2(ADR(str), ADR(comma), ADR(str), SIZEOF(str));
			ELSE
				CONCAT2(ADR(str), ADR(arrayEnd2), ADR(str), SIZEOF(str));
			END_IF
			
		END_FOR
		
		CONCAT2(ADR(sPayloadPub), ADR(str), ADR(sPayloadPub), SIZEOF(sPayloadPub));
		
		(* payload lead string *)
		str	:= ',"payload_lead":[';
		FOR i:=1 TO Get_Data.Data_Length BY 1 DO
			CONCAT2(ADR(str), ADR(Get_Data.Payload_Lead[i]), ADR(str), SIZEOF(str)); 
			
			IF i <> Get_Data.Data_Length THEN
				CONCAT2(ADR(str), ADR(comma), ADR(str), SIZEOF(str));
			ELSE
				CONCAT2(ADR(str), ADR(arrayEnd2), ADR(str), SIZEOF(str));
			END_IF
			
		END_FOR
		
		CONCAT2(ADR(sPayloadPub), ADR(str), ADR(sPayloadPub), SIZEOF(sPayloadPub));
		
		(* payload rear string *)
		str	:= ',"payload_rear":[';
		FOR i:=1 TO Get_Data.Data_Length BY 1 DO
			CONCAT2(ADR(str), ADR(Get_Data.Payload_Rear[i]), ADR(str), SIZEOF(str)); 
			
			IF i <> Get_Data.Data_Length THEN
				CONCAT2(ADR(str), ADR(comma), ADR(str), SIZEOF(str));
			ELSE
				CONCAT2(ADR(str), ADR(arrayEnd2), ADR(str), SIZEOF(str));
			END_IF
			
		END_FOR
		
		CONCAT2(ADR(sPayloadPub), ADR(str), ADR(sPayloadPub), SIZEOF(sPayloadPub));
		
		(* overload lead string *)
		str	:= ',"overload_lead":[';
		FOR i:=1 TO Get_Data.Data_Length BY 1 DO
			CONCAT2(ADR(str), ADR(Get_Data.Overload_Lead[i]), ADR(str), SIZEOF(str)); 
			
			IF i <> Get_Data.Data_Length THEN
				CONCAT2(ADR(str), ADR(comma), ADR(str), SIZEOF(str));
			ELSE
				CONCAT2(ADR(str), ADR(arrayEnd2), ADR(str), SIZEOF(str));
			END_IF
			
		END_FOR
		
		CONCAT2(ADR(sPayloadPub), ADR(str), ADR(sPayloadPub), SIZEOF(sPayloadPub));
		
		(* overload rear string *)
		str	:= ',"overload_rear":[';
		FOR i:=1 TO Get_Data.Data_Length BY 1 DO
			CONCAT2(ADR(str), ADR(Get_Data.Overload_Rear[i]), ADR(str), SIZEOF(str)); 
			
			IF i <> Get_Data.Data_Length THEN
				CONCAT2(ADR(str), ADR(comma), ADR(str), SIZEOF(str));
			ELSE
				CONCAT2(ADR(str), ADR(arrayEnd2), ADR(str), SIZEOF(str));
			END_IF
			
		END_FOR
		
		CONCAT2(ADR(sPayloadPub), ADR(str), ADR(sPayloadPub), SIZEOF(sPayloadPub));
		
		(* pressure lead string *)
		str	:= ',"pressure_lead":[';
		FOR i:=1 TO Get_Data.Data_Length BY 1 DO
			CONCAT2(ADR(str), ADR(Get_Data.Pressure_Lead[i]), ADR(str), SIZEOF(str)); 
			
			IF i <> Get_Data.Data_Length THEN
				CONCAT2(ADR(str), ADR(comma), ADR(str), SIZEOF(str));
			ELSE
				CONCAT2(ADR(str), ADR(arrayEnd2), ADR(str), SIZEOF(str));
			END_IF
			
		END_FOR
		
		CONCAT2(ADR(sPayloadPub), ADR(str), ADR(sPayloadPub), SIZEOF(sPayloadPub));
	
		(* pressure rear string *)
		str	:= ',"pressure_rear":[';
		FOR i:=1 TO Get_Data.Data_Length BY 1 DO
			CONCAT2(ADR(str), ADR(Get_Data.Pressure_Rear[i]), ADR(str), SIZEOF(str)); 
			
			IF i <> Get_Data.Data_Length THEN
				CONCAT2(ADR(str), ADR(comma), ADR(str), SIZEOF(str));
			ELSE
				CONCAT2(ADR(str), ADR(arrayEnd2), ADR(str), SIZEOF(str));
			END_IF
			
		END_FOR
		
		CONCAT2(ADR(sPayloadPub), ADR(str), ADR(sPayloadPub), SIZEOF(sPayloadPub));
		
		(* overpressure lead string *)
		str	:= ',"overpressure_lead":[';
		FOR i:=1 TO Get_Data.Data_Length BY 1 DO
			CONCAT2(ADR(str), ADR(Get_Data.Overpressure_Lead[i]), ADR(str), SIZEOF(str)); 
			
			IF i <> Get_Data.Data_Length THEN
				CONCAT2(ADR(str), ADR(comma), ADR(str), SIZEOF(str));
			ELSE
				CONCAT2(ADR(str), ADR(arrayEnd2), ADR(str), SIZEOF(str));
			END_IF
			
		END_FOR
		
		CONCAT2(ADR(sPayloadPub), ADR(str), ADR(sPayloadPub), SIZEOF(sPayloadPub));
		
		(* overpressure rear string *)
		str	:= ',"overpressure_rear":[';
		FOR i:=1 TO Get_Data.Data_Length BY 1 DO
			CONCAT2(ADR(str), ADR(Get_Data.Overpressure_Rear[i]), ADR(str), SIZEOF(str)); 
			
			IF i <> Get_Data.Data_Length THEN
				CONCAT2(ADR(str), ADR(comma), ADR(str), SIZEOF(str));
			ELSE
				CONCAT2(ADR(str), ADR(arrayEnd2), ADR(str), SIZEOF(str));
			END_IF
			
		END_FOR
		
		CONCAT2(ADR(sPayloadPub), ADR(str), ADR(sPayloadPub), SIZEOF(sPayloadPub));
		
		(* event code string *)
		str	:= ',"event_code":[';
		FOR i:=1 TO Get_Data.Data_Length BY 1 DO
			CONCAT2(ADR(str), ADR(Get_Data.EventCode[i]), ADR(str), SIZEOF(str)); 
			
			IF i <> Get_Data.Data_Length THEN
				CONCAT2(ADR(str), ADR(comma), ADR(str), SIZEOF(str));
			ELSE
				CONCAT2(ADR(str), ADR(arrayEnd2), ADR(str), SIZEOF(str));
			END_IF
			
		END_FOR
		
		CONCAT2(ADR(sPayloadPub), ADR(str), ADR(sPayloadPub), SIZEOF(sPayloadPub));
		
		CONCAT2(ADR(sPayloadPub), ADR(msgEnd), ADR(sPayloadPub), SIZEOF(sPayloadPub)); //message ending
		
		(* publish message to subscribed topic *)
		IF Publish_Data := fbMqttClient.Publish(sTopic:= sTopicPub, pPayload:= ADR(sPayloadPub), nPayloadSize:= LEN2(ADR(sPayloadPub)), eQoS:= TcIotMqttQos.AtMostOnceDelivery, bRetain:= FALSE, bQueue:= FALSE) THEN
			IF fbMqttClient.bError THEN
				// add your error logging here			
				hrErrorOccurred := fbMqttClient.hrErrorCode;
			ELSE
				Published_Data 	:= TRUE;
			END_IF
			
		END_IF
		
	END_IF
	
END_IF

(* send imu *)
IF Main_Send.New_IMU THEN
	Publish_IMU		:= FALSE;
	Published_IMU 	:= FALSE;

	IF fbMqttClient.bConnected THEN	
		IF NOT bSubscribed THEN
			bSubscribed := fbMqttClient.Subscribe(sTopic:=sTopicSub_2, eQoS:=TcIotMqttQos.AtMostOnceDelivery); //subscribe to topic
			IF fbMqttClient.bError THEN
				// add your error logging here
				hrErrorOccurred := fbMqttClient.hrErrorCode;
			END_IF
		END_IF
		
		(* build message payload *)
		sPayloadPub := CONCAT('{"primemover_id":', Read_ID.PrimeMover_ID);
		
		(* lead trailer id string *)
		str	:= ',"trailer_id_lead":[';
		FOR i:=1 TO Get_IMU.Data_Length BY 1 DO
			CONCAT2(ADR(str), ADR(Get_IMU.Trailer_ID_Lead[i]), ADR(str), SIZEOF(str)); 
			
			IF i <> Get_IMU.Data_Length THEN
				CONCAT2(ADR(str), ADR(comma), ADR(str), SIZEOF(str));
			ELSE
				CONCAT2(ADR(str), ADR(arrayEnd2), ADR(str), SIZEOF(str));
			END_IF
			
		END_FOR
		
		CONCAT2(ADR(sPayloadPub), ADR(str), ADR(sPayloadPub), SIZEOF(sPayloadPub));
		
		(* rear trailer id string *)
		str	:= ',"trailer_id_rear":[';
		FOR i:=1 TO Get_IMU.Data_Length BY 1 DO
			CONCAT2(ADR(str), ADR(Get_IMU.Trailer_ID_Rear[i]), ADR(str), SIZEOF(str)); 
			
			IF i <> Get_IMU.Data_Length THEN
				CONCAT2(ADR(str), ADR(comma), ADR(str), SIZEOF(str));
			ELSE
				CONCAT2(ADR(str), ADR(arrayEnd2), ADR(str), SIZEOF(str));
			END_IF
			
		END_FOR
		
		CONCAT2(ADR(sPayloadPub), ADR(str), ADR(sPayloadPub), SIZEOF(sPayloadPub));
		
		(* date time string *)
		str	:= ',"datetime":["';
		FOR i:=1 TO Get_IMU.Data_Length BY 1 DO
			CONCAT2(ADR(str), ADR(Get_IMU.TimeStr[i]), ADR(str), SIZEOF(str)); 
			
			IF i <> Get_IMU.Data_Length THEN
				CONCAT2(ADR(str), ADR(valSeparator), ADR(str), SIZEOF(str));
			ELSE
				CONCAT2(ADR(str), ADR(arrayEnd), ADR(str), SIZEOF(str));
			END_IF
			
		END_FOR
		
		CONCAT2(ADR(sPayloadPub), ADR(str), ADR(sPayloadPub), SIZEOF(sPayloadPub));
		
		(* lead pitch string *)
		str	:= ',"pitch_lead":[';
		FOR i:=1 TO Get_IMU.Data_Length BY 1 DO
			CONCAT2(ADR(str), ADR(Get_IMU.Pitch_Lead[i]), ADR(str), SIZEOF(str)); 
			
			IF i <> Get_IMU.Data_Length THEN
				CONCAT2(ADR(str), ADR(comma), ADR(str), SIZEOF(str));
			ELSE
				CONCAT2(ADR(str), ADR(arrayEnd2), ADR(str), SIZEOF(str));
			END_IF
			
		END_FOR
		
		CONCAT2(ADR(sPayloadPub), ADR(str), ADR(sPayloadPub), SIZEOF(sPayloadPub));
		
		(* lead roll string *)
		str	:= ',"roll_lead":[';
		FOR i:=1 TO Get_IMU.Data_Length BY 1 DO
			CONCAT2(ADR(str), ADR(Get_IMU.Roll_Lead[i]), ADR(str), SIZEOF(str)); 
			
			IF i <> Get_IMU.Data_Length THEN
				CONCAT2(ADR(str), ADR(comma), ADR(str), SIZEOF(str));
			ELSE
				CONCAT2(ADR(str), ADR(arrayEnd2), ADR(str), SIZEOF(str));
			END_IF
			
		END_FOR
		
		CONCAT2(ADR(sPayloadPub), ADR(str), ADR(sPayloadPub), SIZEOF(sPayloadPub));
		
		(* lead acceleration x string *)
		str	:= ',"ax_lead":[';
		FOR i:=1 TO Get_IMU.Data_Length BY 1 DO
			CONCAT2(ADR(str), ADR(Get_IMU.AccX_Lead[i]), ADR(str), SIZEOF(str)); 
			
			IF i <> Get_IMU.Data_Length THEN
				CONCAT2(ADR(str), ADR(comma), ADR(str), SIZEOF(str));
			ELSE
				CONCAT2(ADR(str), ADR(arrayEnd2), ADR(str), SIZEOF(str));
			END_IF
			
		END_FOR
		
		CONCAT2(ADR(sPayloadPub), ADR(str), ADR(sPayloadPub), SIZEOF(sPayloadPub));
		
		(* lead acceleration y string *)
		str	:= ',"ay_lead":[';
		FOR i:=1 TO Get_IMU.Data_Length BY 1 DO
			CONCAT2(ADR(str), ADR(Get_IMU.AccY_Lead[i]), ADR(str), SIZEOF(str)); 
			
			IF i <> Get_IMU.Data_Length THEN
				CONCAT2(ADR(str), ADR(comma), ADR(str), SIZEOF(str));
			ELSE
				CONCAT2(ADR(str), ADR(arrayEnd2), ADR(str), SIZEOF(str));
			END_IF
			
		END_FOR
		
		CONCAT2(ADR(sPayloadPub), ADR(str), ADR(sPayloadPub), SIZEOF(sPayloadPub));
		
		(* lead acceleration z string *)
		str	:= ',"az_lead":[';
		FOR i:=1 TO Get_IMU.Data_Length BY 1 DO
			CONCAT2(ADR(str), ADR(Get_IMU.AccZ_Lead[i]), ADR(str), SIZEOF(str)); 
			
			IF i <> Get_IMU.Data_Length THEN
				CONCAT2(ADR(str), ADR(comma), ADR(str), SIZEOF(str));
			ELSE
				CONCAT2(ADR(str), ADR(arrayEnd2), ADR(str), SIZEOF(str));
			END_IF
			
		END_FOR
		
		CONCAT2(ADR(sPayloadPub), ADR(str), ADR(sPayloadPub), SIZEOF(sPayloadPub));
		
		(* lead pitch string *)
		str	:= ',"pitch_rear":[';
		FOR i:=1 TO Get_IMU.Data_Length BY 1 DO
			CONCAT2(ADR(str), ADR(Get_IMU.Pitch_Rear[i]), ADR(str), SIZEOF(str)); 
			
			IF i <> Get_IMU.Data_Length THEN
				CONCAT2(ADR(str), ADR(comma), ADR(str), SIZEOF(str));
			ELSE
				CONCAT2(ADR(str), ADR(arrayEnd2), ADR(str), SIZEOF(str));
			END_IF
			
		END_FOR
		
		CONCAT2(ADR(sPayloadPub), ADR(str), ADR(sPayloadPub), SIZEOF(sPayloadPub));
		
		(* rear roll string *)
		str	:= ',"roll_rear":[';
		FOR i:=1 TO Get_IMU.Data_Length BY 1 DO
			CONCAT2(ADR(str), ADR(Get_IMU.Roll_Rear[i]), ADR(str), SIZEOF(str)); 
			
			IF i <> Get_IMU.Data_Length THEN
				CONCAT2(ADR(str), ADR(comma), ADR(str), SIZEOF(str));
			ELSE
				CONCAT2(ADR(str), ADR(arrayEnd2), ADR(str), SIZEOF(str));
			END_IF
			
		END_FOR
		
		CONCAT2(ADR(sPayloadPub), ADR(str), ADR(sPayloadPub), SIZEOF(sPayloadPub));
		
		(* rear acceleration x string *)
		str	:= ',"ax_rear":[';
		FOR i:=1 TO Get_IMU.Data_Length BY 1 DO
			CONCAT2(ADR(str), ADR(Get_IMU.AccX_Rear[i]), ADR(str), SIZEOF(str)); 
			
			IF i <> Get_IMU.Data_Length THEN
				CONCAT2(ADR(str), ADR(comma), ADR(str), SIZEOF(str));
			ELSE
				CONCAT2(ADR(str), ADR(arrayEnd2), ADR(str), SIZEOF(str));
			END_IF
			
		END_FOR
		
		CONCAT2(ADR(sPayloadPub), ADR(str), ADR(sPayloadPub), SIZEOF(sPayloadPub));
		
		(* rear acceleration y string *)
		str	:= ',"ay_rear":[';
		FOR i:=1 TO Get_IMU.Data_Length BY 1 DO
			CONCAT2(ADR(str), ADR(Get_IMU.AccY_Rear[i]), ADR(str), SIZEOF(str)); 
			
			IF i <> Get_IMU.Data_Length THEN
				CONCAT2(ADR(str), ADR(comma), ADR(str), SIZEOF(str));
			ELSE
				CONCAT2(ADR(str), ADR(arrayEnd2), ADR(str), SIZEOF(str));
			END_IF
			
		END_FOR
		
		CONCAT2(ADR(sPayloadPub), ADR(str), ADR(sPayloadPub), SIZEOF(sPayloadPub));
		
		(* rear acceleration z string *)
		str	:= ',"az_rear":[';
		FOR i:=1 TO Get_IMU.Data_Length BY 1 DO
			CONCAT2(ADR(str), ADR(Get_IMU.AccZ_Rear[i]), ADR(str), SIZEOF(str)); 
			
			IF i <> Get_IMU.Data_Length THEN
				CONCAT2(ADR(str), ADR(comma), ADR(str), SIZEOF(str));
			ELSE
				CONCAT2(ADR(str), ADR(arrayEnd2), ADR(str), SIZEOF(str));
			END_IF
			
		END_FOR
		
		CONCAT2(ADR(sPayloadPub), ADR(str), ADR(sPayloadPub), SIZEOF(sPayloadPub));
		
		CONCAT2(ADR(sPayloadPub), ADR(msgEnd), ADR(sPayloadPub), SIZEOF(sPayloadPub)); //message ending
		
		(* publish message to subscribed topic *)
		IF Publish_IMU := fbMqttClient.Publish(sTopic:= sTopicPub_2, pPayload:= ADR(sPayloadPub), nPayloadSize:= LEN2(ADR(sPayloadPub)), eQoS:= TcIotMqttQos.AtMostOnceDelivery, bRetain:= FALSE, bQueue:= FALSE) THEN
			IF fbMqttClient.bError THEN
				// add your error logging here			
				hrErrorOccurred := fbMqttClient.hrErrorCode;
			ELSE
				Published_IMU 	:= TRUE;
			END_IF
			
		END_IF
		
	END_IF	
END_IF

END_PROGRAM

// ---- POUs/Read_ID.TcPOU
PROGRAM Read_ID
VAR
	PrimeMover_ID			: STRING := '2';
	Trailer_ID_Lead AT %I*	: UINT;
	Trailer_ID_Rear AT %I*	: UINT;
END_VAR

;

END_PROGRAM

// ---- POUs/Main_Vacuum.TcPOU
PROGRAM Main_Vacuum
VAR
END_VAR

IF NOT Vacuum_Buffer_Data.Vacuumed THEN
	Vacuum_Buffer_Data();
END_IF

IF NOT Vacuum_Buffer_Data_2.Vacuumed THEN
	Vacuum_Buffer_Data_2();
END_IF

IF NOT Vacuum_Buffer_IMU.Vacuumed THEN
	Vacuum_Buffer_IMU();
END_IF

IF NOT Vacuum_Buffer_IMU_2.Vacuumed THEN
	Vacuum_Buffer_IMU_2();
END_IF

IF NOT Vacuum_Data.Vacuumed THEN
	Vacuum_Data();
END_IF

IF NOT Vacuum_IMU.Vacuumed THEN
	Vacuum_IMU();
END_IF

END_PROGRAM

// ---- POUs/Vacuum_Buffer_Data.TcPOU
PROGRAM Vacuum_Buffer_Data
VAR
	fbSqlDatabase	: FB_SQLDatabaseEvt(sNetID := '', tTimeout := T#1000S);
	fbSqlCommand	: FB_SQLCommandEvt(sNetID := '', tTimeout := T#1000S);
	fbSqlResult		: FB_SQLResultEvt(sNetID :='', tTimeout   := T#1000S); 
	nState			: INT;
	sCmd			: STRING(500000);
	Vacuumed		: BOOL;
END_VAR

CASE nState OF
				
		0:
			(* connect to buffer_imu *)		
			IF fbSqlDatabase.Connect(1) THEN
				IF fbSqlDatabase.bError THEN
					nState := 255; 
				ELSE
					IF fbSqlDatabase.bConnected THEN
						nState := nState+1;
					END_IF 
				END_IF
			END_IF
			
		1:
			IF fbSqlDatabase.CreateCmd(ADR(fbSqlCommand)) THEN
				IF fbSqlDatabase.bError THEN
					nState := 255; 
				ELSE
					nState := nState+1; 
				END_IF
			END_IF
			
		2:	(* execute pragmas *)
			sCmd	:= 'PRAGMA journal_mode = WAL; PRAGMA synchronous = NORMAL; PRAGMA temp_store = MEMORY; PRAGMA mmap_size = 30000000000; PRAGMA page_size = 32768; PRAGMA locking_mode = EXCLUSIVE;';
			
			IF fbSQLCommand.Execute(ADR(sCmd), SIZEOF(sCmd)) THEN
				IF fbSQLCommand.bError THEN
					nState := 255; 
				ELSE
					nState := nState+1; 
				END_IF
			END_IF
		
		3:	
			IF NOT Vacuumed THEN
				(* build query *)	
				sCmd	:= 'VACUUM';
				
				IF fbSQLCommand.Execute(ADR(sCmd), SIZEOF(sCmd)) THEN
					IF fbSQLCommand.bError THEN
						nState := 255; 
					ELSE
						nState 		:= nState+1; 
					END_IF
				END_IF
				
			ELSE 
				nState := nState+1;
			END_IF
			
		4:	(* execute pragma optimize *)
			sCmd	:= 'PRAGMA optimize;';
			
			IF fbSQLCommand.Execute(ADR(sCmd), SIZEOF(sCmd)) THEN
				IF fbSQLCommand.bError THEN
					nState := 255; 
				ELSE
					nState := nState+1; 
				END_IF
			END_IF
		
		5:
			IF fbSqlDatabase.Disconnect() THEN
				IF fbSqlDatabase.bError THEN
					nState := 255;
				ELSE
					nState 		:= nState+1;
					Vacuumed 	:= TRUE;
				END_IF
			END_IF
			
		255:
			nState := 0;
			
END_CASE

END_PROGRAM

// ---- POUs/Vacuum_Buffer_Data_2.TcPOU
PROGRAM Vacuum_Buffer_Data_2
VAR
	fbSqlDatabase	: FB_SQLDatabaseEvt(sNetID := '', tTimeout := T#1000S);
	fbSqlCommand	: FB_SQLCommandEvt(sNetID := '', tTimeout := T#1000S);
	fbSqlResult		: FB_SQLResultEvt(sNetID :='', tTimeout   := T#1000S); 
	nState			: INT;
	sCmd			: STRING(500000);
	Vacuumed		: BOOL;
END_VAR

CASE nState OF
				
		0:
			(* connect to buffer_imu *)		
			IF fbSqlDatabase.Connect(6) THEN
				IF fbSqlDatabase.bError THEN
					nState := 255; 
				ELSE
					IF fbSqlDatabase.bConnected THEN
						nState := nState+1;
					END_IF 
				END_IF
			END_IF
			
		1:
			IF fbSqlDatabase.CreateCmd(ADR(fbSqlCommand)) THEN
				IF fbSqlDatabase.bError THEN
					nState := 255; 
				ELSE
					nState := nState+1; 
				END_IF
			END_IF
			
		2:	(* execute pragmas *)
			sCmd	:= 'PRAGMA journal_mode = WAL; PRAGMA synchronous = NORMAL; PRAGMA temp_store = MEMORY; PRAGMA mmap_size = 30000000000; PRAGMA page_size = 32768; PRAGMA locking_mode = EXCLUSIVE;';
			
			IF fbSQLCommand.Execute(ADR(sCmd), SIZEOF(sCmd)) THEN
				IF fbSQLCommand.bError THEN
					nState := 255; 
				ELSE
					nState := nState+1; 
				END_IF
			END_IF
		
		3:	
			IF NOT Vacuumed THEN
				(* build query *)	
				sCmd	:= 'VACUUM';
				
				IF fbSQLCommand.Execute(ADR(sCmd), SIZEOF(sCmd)) THEN
					IF fbSQLCommand.bError THEN
						nState := 255; 
					ELSE
						nState 		:= nState+1; 
					END_IF
				END_IF
				
			ELSE 
				nState := nState+1;
			END_IF
			
		4:	(* execute pragma optimize *)
			sCmd	:= 'PRAGMA optimize;';
			
			IF fbSQLCommand.Execute(ADR(sCmd), SIZEOF(sCmd)) THEN
				IF fbSQLCommand.bError THEN
					nState := 255; 
				ELSE
					nState := nState+1; 
				END_IF
			END_IF
		
		5:
			IF fbSqlDatabase.Disconnect() THEN
				IF fbSqlDatabase.bError THEN
					nState := 255;
				ELSE
					nState 		:= nState+1;
					Vacuumed 	:= TRUE;
				END_IF
			END_IF
			
		255:
			nState := 0;
			
END_CASE

END_PROGRAM

// ---- POUs/Background_GPS.TcPOU
PROGRAM Background_GPS

VAR
	RxBuffer	:ComBuffer;
	TxBuffer	:ComBuffer;
	
	fbLineCtrlAds	: SerialLineControlADS;
	bAdsError		: BOOL;
	nAdsErrorID		: UDINT;
	bConnect		: BOOL := TRUE;
	sNetID			: T_amsNetId;
	stSerialCfg		: ComSerialConfig;
	Port			: BOOL;
END_VAR

stSerialCfg.Baudrate := 4800;
stSerialCfg.ComPort := 4;
stSerialCfg.DataBits := 8;
stSerialCfg.Parity := PARITY_NONE;
stSerialCfg.StopBits := STOPBITS_ONE;

fbLineCtrlAds(
	Connect 	:= bConnect,
	SerialCfg	:= stSerialCfg,
	NetId		:= sNetId,
	Timeout		:= T#5s,
	TxBuffer	:= TxBuffer,
	RxBuffer	:= RxBuffer,
	Busy		:= ,
	Error		=> bAdsError,
	ErrorID		=> nAdsErrorID,
	PortOpened	=> Port
);

END_PROGRAM

// ---- POUs/FB_FatigueCam_Receive.TcPOU
	FUNCTION_BLOCK FB_FatigueCam_Receive

VAR_IN_OUT
	RxBuffer	: ComBuffer;
END_VAR

VAR_INPUT
	Command		: ULINT;
	Prefix		: WORD;
	LenPrefix	: BYTE;
END_VAR

VAR_OUTPUT
	Response	: STRING;
	EventCode	: STRING;
	EventID		: STRING;
	//TimeSync	: STRING;
END_VAR

VAR
	fbReceive		: ReceiveData;
	bReceiveBusy	: BOOL;
	bReceiveError	: BOOL;
	eReceiveErrorID	: ComError_t;
	bReceiveTimeout	: BOOL;
	nReceiveCounter	: UDINT;
	receive			: ULINT;
	bDataReceived	: BOOL;
	bSend			: BOOL;
	bSend1			: BOOL;
	fbClearCom		: ClearComBuffer;
	
	//Response		: STRING;
	InstructionID	: STRING;
	
	bEventID		: BYTE;
	prevEventID		: STRING;
	FatigueCode		: STRING;
	AbnormCode		: STRING;
END_VAR

(* receive data *)
fbReceive( 
	RxBuffer := RxBuffer,
	pPrefix := ADR(Prefix),
	LenPrefix := LenPrefix,
	pReceiveData := ADR(receive),
	SizeReceiveData	:= 6,
	Timeout:= T#1S,
	Busy => bReceiveBusy,
	Error => ,
	DataReceived => bDataReceived,
	RxTimeout=> bReceiveTimeout 
);

IF fbReceive.Error <> COMERROR_NOERROR THEN
	eReceiveErrorID := fbReceive.Error;
END_IF
IF bDataReceived THEN
	nReceiveCounter := nReceiveCounter + 1;
END_IF

(* response parsing *)
Response 		:= LWORD_TO_HEXSTR(in := receive, iPrecision := 16, bLoCase := FALSE);
InstructionID	:= RIGHT(STR := Response, SIZE := 4);
IF InstructionID = '8BAA' THEN
	EventID		:= MID(STR := Response, LEN := 2, POS := 7);
	HEXSTR_TO_DATA(EventID, ADR(bEventID), SIZEOF(bEventID)); 
	EventID		:= BYTE_TO_DECSTR(in := bEventID, iPrecision := 1);
	
	AbnormCode	:= MID(STR := Response, LEN := 2, POS := 9);
	FatigueCode	:= MID(STR := Response, LEN := 2, POS := 11);
	
	(* event classification *)
	IF EventID <> prevEventID THEN
		IF FatigueCode = '00' AND AbnormCode = '00' THEN
			EventCode	:= '0'; //no events
		ELSIF FatigueCode = '01' THEN
			EventCode	:= '1'; //lv 1 fatigue
		ELSIF FatigueCode = '02' THEN
			EventCode	:= '2'; //lv 2 fatigue
		ELSIF FatigueCode = '03' THEN
			EventCode	:= '3'; //smoking
		ELSIF FatigueCode = '04' THEN
			EventCode	:= '4'; //phone
		ELSIF FatigueCode = '05' THEN
			EventCode	:= '5'; //head down
		ELSIF FatigueCode = '06' THEN
			EventCode	:= '6'; //yawn
		ELSIF FatigueCode = '07' THEN
			EventCode	:= '7'; //look around
		ELSIF FatigueCode = '08' THEN
			EventCode	:= '8'; //chat
		ELSIF AbnormCode = '02' THEN
			EventCode	:= '9'; //face missing
		ELSIF AbnormCode = '10' THEN
			EventCode	:= '10'; //camera covered
		END_IF
		prevEventID	:= EventID;
	END_IF
END_IF

(* error handling *)
//IF InstructionID = '8FAA' THEN
//END_IF

fbClearCom(Buffer := RxBuffer); //clear rx buffer

END_FUNCTION_BLOCK

// ---- POUs/Read_Pressure.TcPOU
PROGRAM Read_Pressure
VAR
	EL3052_Lead_Bit AT %I* : INT;
	EL3052_Rear_Bit AT %I* : INT;
	
	Pressure_Lead		: REAL;
	Pressure_Rear		: REAL;
	Threshold			: REAL := 180;
	
	Overpressure_Lead	: BOOL;
	Overpressure_Rear	: BOOL;
	
END_VAR

(* read pressure *)
IF GVL.Lead_Trailer_State = 8 OR GVL.Lead_Trailer_State = 17416 THEN
	Pressure_Lead 	:= (INT_TO_REAL(EL3052_Lead_Bit)/32767) * 160;
ELSE
	Pressure_Lead 	:= 0;	
END_IF

IF GVL.Rear_Trailer_State = 8 THEN
	Pressure_Rear 	:= (INT_TO_REAL(EL3052_Rear_Bit)/32767) * 160;
ELSE
	Pressure_Rear 	:= 0;
END_IF

(* check for overpressure *)
IF Pressure_Lead > Threshold THEN
	Overpressure_Lead := TRUE;
ELSE
	Overpressure_Lead := FALSE;
END_IF

IF Pressure_Rear > Threshold THEN
	Overpressure_Rear := TRUE;
ELSE
	Overpressure_Rear := FALSE;
END_IF

(* only read over pressure event once during dump cycle *)

END_PROGRAM

// ---- POUs/Read_Payload.TcPOU
PROGRAM Read_Payload
VAR
	EL3061_Lead_Bit AT %I* 	: INT;
	EL3061_Rear_Bit AT %I* 	: INT;
	
	//axle of lead trailer
	R3_Bit			: REAL;
	R3_BitTare		: REAL := 8043;
	R31_BitPerTon	: REAL := 7.8864; //bit caused by payload on lead trailer
	R32_BitPerTon	: REAL := 7.8864; //bit caused by payload on rear trailer
	
	//axle of rear trailer
	R4_Bit			: REAL;
	R4_BitTare		: REAL := 8043;
	R42_BitPerTon	: REAL := 7.8864;
	
	Payload_Lead	: REAL;
	Payload_Rear	: REAL;
	Payload_Total	: REAL;	
	
	Threshold_Lead	: REAL := 40.5;
	Threshold_Rear	: REAL := 72;	
	Overload_Lead	: BOOL := FALSE;
	Overload_Rear	: BOOL := FALSE;
END_VAR

R3_Bit := INT_TO_REAL(EL3061_Lead_Bit);
R4_Bit := INT_TO_REAL(EL3061_Rear_Bit);

(*
Payload_Rear	:= (R4_Bit - R4_BitTare) / R42_BitPerTon;
Payload_Lead	:= (R3_Bit - (R32_BitPerTon * Payload_Rear)) / R31_BitPerTon;
Payload_Total	:= Payload_Lead + Payload_Rear;
*)

//Payload_Rear	:= (R4_Bit - R4_BitTare) / R42_BitPerTon;

IF GVL.Lead_Trailer_State = 8 OR GVL.Lead_Trailer_State = 17416 THEN
	Payload_Lead	:= R3_Bit;
ELSE
	Payload_Lead	:= 0;
END_IF

IF GVL.Rear_Trailer_State = 8 THEN
	Payload_Rear	:= R4_Bit;
ELSE
	Payload_Rear	:= 0;
END_IF
Payload_Rear	:= R4_Bit;

IF Payload_Lead < 0 THEN
	Payload_Lead := 0;
END_IF

IF Payload_Rear < 0 THEN
	Payload_Rear := 0;
END_IF

IF Payload_Lead > Threshold_Lead THEN
	Overload_Lead := TRUE;
ELSE
	Overload_Lead := FALSE;	
END_IF

IF Payload_Rear > Threshold_Rear THEN
	Overload_Rear := TRUE;
ELSE
	Overload_Rear := FALSE;	
END_IF

(*
IF Read_GPS.Speed < 1 AND Background_IMU.Pitch < 3 AND Background_IMU.Roll < 3 THEN
	Payload	:= Payload_Raw;
END_IF

(* check for overload *)
IF Payload > Threshold THEN
	Overload := TRUE;
ELSE
	Overload := FALSE;	
END_IF
*)

END_PROGRAM

// ---- POUs/Read_GPS.TcPOU
PROGRAM Read_GPS
VAR
	(* receive string variables *)
	fbReceiveString	: ReceiveString;
	DataString		: STRING;
	Pref			: STRING := '$$GPRMC,';
	Suff			: STRING := '*';
	
	(* parsing variables *)
    sSeparator   : STRING(1) := ',';
	sSeparator2  : STRING(1) := '.';
    aSplit       : ARRAY[1..cMax] OF STRING; //parsed string
    bResultSplit : BOOL;
    i            : UDINT;
	
	(* gps variables *)
	HourInt		: INT;
	HourStr		: STRING;
	TimeStamp	: STRING;
	LatLeftStr	: STRING;
	LatRightStr	: STRING;
	LonLeftStr	: STRING;
	LonRightStr	: STRING;
	LatLeft		: INT;
	LatRight	: INT;
	LonLeft		: INT;
	LonRight	: INT;
	LatDeg		: REAL;
	LonDeg		: REAL;
	LatMin		: REAL;
	LonMin		: REAL;
	Lat			: REAL;
	Lon			: REAL;
	Speed		: REAL;
	Threshold	: REAL := 60;
	Overspeed	: BOOL := FALSE;
	
	Cycle_Duration	: STRING := '0';
	
	pSec	: WORD;
END_VAR

VAR CONSTANT
    cMax         : UDINT := 11; //no. of substrings
END_VAR

(* get gps data string *)
fbReceiveString(
	RxBuffer := Background_GPS.RxBuffer, 
	Prefix := Pref, 
	Suffix := Suff, 
	Timeout := T#1S, 
	ReceivedString := DataString
);

(* gps data parsing *)
aSplit[1] := DataString;
FOR i:=1 TO cMax-1 DO
	bResultSplit := FindAndSplit( 
						pSeparator     := ADR(sSeparator),  
						pSrcString := ADR(aSplit[i]), 
						pLeftString    := ADR(aSplit[i]),   
						nLeftSize  := SIZEOF(aSplit[i]), 
						pRightString   := ADR(aSplit[i+1]), 
						nRightSize := SIZEOF(aSplit[i+1]),
						bSearchFromRight := FALSE 
					);
	IF NOT bResultSplit THEN
		EXIT;
	END_IF
END_FOR

IF aSplit[3] = 'A' THEN
	(* latitude & longitude conversion *)
	FindAndSplit( 
		pSeparator     		:= ADR(sSeparator2),  
		pSrcString 			:= ADR(aSplit[4]), 
		pLeftString    		:= ADR(LatLeftStr),   
		nLeftSize  			:= SIZEOF(LatLeftStr), 
		pRightString   		:= ADR(LatRightStr), 
		nRightSize 			:= SIZEOF(LatRightStr),
		bSearchFromRight 	:= FALSE 
	);
	
	FindAndSplit( 
		pSeparator     		:= ADR(sSeparator2),  
		pSrcString 			:= ADR(aSplit[6]), 
		pLeftString    		:= ADR(LonLeftStr),   
		nLeftSize  			:= SIZEOF(LonLeftStr), 
		pRightString   		:= ADR(LonRightStr), 
		nRightSize 			:= SIZEOF(LonRightStr),
		bSearchFromRight 	:= FALSE 
	);
	
	LatLeft 	:= STRING_TO_INT(LatLeftStr);
	LatRight 	:= STRING_TO_INT(LatRightStr);
	LonLeft 	:= STRING_TO_INT(LonLeftStr);
	LonRight 	:= STRING_TO_INT(LonRightStr);
	Lat			:= INT_TO_REAL(LatLeft) + (INT_TO_REAL(LatRight)/EXPT(10,LEN(LatRightStr)));
	Lon 		:= INT_TO_REAL(LonLeft) + (INT_TO_REAL(LonRight)/EXPT(10,LEN(LonRightStr)));;
	LatDeg 		:= TRUNC(Lat/100);
	LonDeg 		:= TRUNC(Lon/100);
	LatMin 		:= Lat - (LatDeg*100);
	LonMin 		:= Lon - (LonDeg*100);
	Lat 		:= LatDeg + (LatMin/60);
	Lon			:= LonDeg + (LonMin/60);
	
	IF aSplit[5] = 'S' THEN
		Lat := Lat*(-1);
	END_IF
	
	IF aSplit[7] = 'W' THEN
		Lon := Lon*(-1); 
	END_IF
	
	(* speed conversion *)
	Speed	:= STRING_TO_REAL(aSplit[8]) * 1.852;

ELSE
	(* gps no signal error handling *)
END_IF

(* check for overspeed *)
IF Speed > Threshold THEN
	Overspeed := TRUE;
ELSE
	Overspeed := FALSE;
END_IF

END_PROGRAM

// ---- POUs/Send_IMU.TcPOU
PROGRAM Send_IMU
VAR
	fbMqttClient : FB_IotMqttClient;
	bSetParameter : BOOL := TRUE;
	bConnect : BOOL := TRUE;
	
	(* aws certificates *)
	
	(*-------------- actual ------------------*)
	(*
	rootCA		: STRING(255) := 'C:\Users\Administrator\Downloads\AWSCert\AmazonRootCA1.pem';
	thingCert	: STRING(255) := 'C:\Users\Administrator\Downloads\AWSCert\a2ca8bd1ed97a43e38f2bffcdf7ca64a29d3483826fdb03b3eb616af8a5efc9e-certificate.pem.crt';
	privateKey	: STRING(255) := 'C:\Users\Administrator\Downloads\AWSCert\a2ca8bd1ed97a43e38f2bffcdf7ca64a29d3483826fdb03b3eb616af8a5efc9e-private.pem.key';
	*)
	
	rootCA		: STRING(255) := 'C:\Users\Administrator\Downloads\AWSCert\AmazonRootCA1.pem';
	thingCert	: STRING(255) := 'C:\Users\Administrator\Downloads\AWSCert\8872c9f9d2c9335079f20c0506a3dd3599fd4d8552622bd2d7f8ae6d1681c64f-certificate.pem.crt';
	privateKey	: STRING(255) := 'C:\Users\Administrator\Downloads\AWSCert\8872c9f9d2c9335079f20c0506a3dd3599fd4d8552622bd2d7f8ae6d1681c64f-private.pem.key';
	
	(* ---------------- test ------------------- *)
	(*
	rootCA		: STRING(255) := 'C:\Users\muhammad.rahman\Downloads\double-sdt-test-certs\AmazonRootCA1.pem';
	thingCert	: STRING(255) := 'C:\Users\muhammad.rahman\Downloads\double-sdt-test-certs\8872c9f9d2c9335079f20c0506a3dd3599fd4d8552622bd2d7f8ae6d1681c64f-certificate.pem.crt';
	privateKey	: STRING(255) := 'C:\Users\muhammad.rahman\Downloads\double-sdt-test-certs\8872c9f9d2c9335079f20c0506a3dd3599fd4d8552622bd2d7f8ae6d1681c64f-private.pem.key';
	*)
	
	(* broker settings *)
	endpoint	: STRING := 'a2o01t3xth0mr1-ats.iot.ap-southeast-1.amazonaws.com';
	port		: UINT := 8883;
	//clientID	: STRING := 'double-sdt-1';
	clientID	: STRING := 'double-sdt-test';
	
	(* published message *)
	sTopicPub 		: STRING(255) := 'iot/smartproduct/mifa/double-sdt/imu'; //message topic
	sPayloadPub 	: STRING(50000000);
	str				: STRING(10000000);
	valSeparator	: STRING := '","';
	comma			: STRING := ',';
	arrayEnd		: STRING := '"]';
	arrayEnd2		: STRING := ']';
	msgEnd			: STRING := '}';
	i				: ULINT;
	
	(* topic subscription *)
	bSubscribed : BOOL;
	sTopicSub 	: STRING(255) := 'iot/smartproduct/mifa/double-sdt/imu';
	
	(* received message *)	
	{attribute 'TcEncoding':='UTF-8'}
	sTopicRcv : STRING(255);
	{attribute 'TcEncoding':='UTF-8'}
	sPayloadRcv : STRING(255);
	
	fbMessageQueue : FB_IotMqttMessageQueue;
	fbMessage : FB_IotMqttMessage;
	
	hrErrorOccurred : HRESULT; // contains the latest occurred error
	Published		: BOOL;
	Publish			: BOOL;
END_VAR

IF Main_SendIMU.New_Data THEN
	Publish		:= FALSE;
	Published 	:= FALSE;	
END_IF


IF bSetParameter THEN
	bSetParameter := FALSE;
	
	(* TLS settings for AWS IoT connection *)
	fbMqttClient.stTLS.sCA 		:= rootCA; //root CA
    fbMqttClient.stTLS.sCert 	:= thingCert; //certificate of thing
    fbMqttClient.stTLS.sKeyFile := privateKey; //private key of thing
	
	(* Broker settings für AWS IoT *)
	fbMqttClient.sHostName:= endpoint; //broker endpoint
	fbMqttClient.nHostPort:= port; //default mqtt tls port
	fbMqttClient.sClientId:= clientID; //client id
	fbMqttClient.sTopicPrefix:= ''; 
	
	fbMqttClient.ipMessageQueue := fbMessageQueue;
END_IF

(* connect to mqtt broker *)
fbMqttClient.Execute(bConnect); 
IF fbMqttClient.bError THEN
	// add your error logging here
	hrErrorOccurred := fbMqttClient.hrErrorCode;
END_IF

(* get message from subscribed topic *)
IF fbMessageQueue.nQueuedMessages > 0 THEN
	IF fbMessageQueue.Dequeue(fbMessage:=fbMessage) THEN
		fbMessage.GetTopic(pTopic:=ADR(sTopicRcv), nTopicSize:=SIZEOF(sTopicRcv) );
		fbMessage.GetPayload(pPayload:=ADR(sPayloadRcv), nPayloadSize:=SIZEOF(sPayloadRcv), bSetNullTermination:=FALSE);
	END_IF
END_IF

IF fbMqttClient.bConnected THEN	
	IF NOT bSubscribed THEN
		bSubscribed := fbMqttClient.Subscribe(sTopic:=sTopicSub, eQoS:=TcIotMqttQos.AtMostOnceDelivery); //subscribe to topic
		IF fbMqttClient.bError THEN
			// add your error logging here
			hrErrorOccurred := fbMqttClient.hrErrorCode;
		END_IF
	END_IF
	
	(* build message payload *)
	sPayloadPub := CONCAT('{"primemover_id":', Read_ID.PrimeMover_ID);
	
	(* lead trailer id string *)
	str	:= ',"trailer_id_lead":[';
	FOR i:=1 TO Get_IMU.Data_Length BY 1 DO
		CONCAT2(ADR(str), ADR(Get_IMU.Trailer_ID_Lead[i]), ADR(str), SIZEOF(str)); 
		
		IF i <> Get_IMU.Data_Length THEN
			CONCAT2(ADR(str), ADR(comma), ADR(str), SIZEOF(str));
		ELSE
			CONCAT2(ADR(str), ADR(arrayEnd2), ADR(str), SIZEOF(str));
		END_IF
		
	END_FOR
	
	CONCAT2(ADR(sPayloadPub), ADR(str), ADR(sPayloadPub), SIZEOF(sPayloadPub));
	
	(* rear trailer id string *)
	str	:= ',"trailer_id_rear":[';
	FOR i:=1 TO Get_IMU.Data_Length BY 1 DO
		CONCAT2(ADR(str), ADR(Get_IMU.Trailer_ID_Rear[i]), ADR(str), SIZEOF(str)); 
		
		IF i <> Get_IMU.Data_Length THEN
			CONCAT2(ADR(str), ADR(comma), ADR(str), SIZEOF(str));
		ELSE
			CONCAT2(ADR(str), ADR(arrayEnd2), ADR(str), SIZEOF(str));
		END_IF
		
	END_FOR
	
	CONCAT2(ADR(sPayloadPub), ADR(str), ADR(sPayloadPub), SIZEOF(sPayloadPub));
	
	(* date time string *)
	str	:= ',"datetime":["';
	FOR i:=1 TO Get_IMU.Data_Length BY 1 DO
		CONCAT2(ADR(str), ADR(Get_IMU.TimeStr[i]), ADR(str), SIZEOF(str)); 
		
		IF i <> Get_IMU.Data_Length THEN
			CONCAT2(ADR(str), ADR(valSeparator), ADR(str), SIZEOF(str));
		ELSE
			CONCAT2(ADR(str), ADR(arrayEnd), ADR(str), SIZEOF(str));
		END_IF
		
	END_FOR
	
	CONCAT2(ADR(sPayloadPub), ADR(str), ADR(sPayloadPub), SIZEOF(sPayloadPub));
	
	(* lead pitch string *)
	str	:= ',"pitch_lead":[';
	FOR i:=1 TO Get_IMU.Data_Length BY 1 DO
		CONCAT2(ADR(str), ADR(Get_IMU.Pitch_Lead[i]), ADR(str), SIZEOF(str)); 
		
		IF i <> Get_IMU.Data_Length THEN
			CONCAT2(ADR(str), ADR(comma), ADR(str), SIZEOF(str));
		ELSE
			CONCAT2(ADR(str), ADR(arrayEnd2), ADR(str), SIZEOF(str));
		END_IF
		
	END_FOR
	
	CONCAT2(ADR(sPayloadPub), ADR(str), ADR(sPayloadPub), SIZEOF(sPayloadPub));
	
	(* lead roll string *)
	str	:= ',"roll_lead":[';
	FOR i:=1 TO Get_IMU.Data_Length BY 1 DO
		CONCAT2(ADR(str), ADR(Get_IMU.Roll_Lead[i]), ADR(str), SIZEOF(str)); 
		
		IF i <> Get_IMU.Data_Length THEN
			CONCAT2(ADR(str), ADR(comma), ADR(str), SIZEOF(str));
		ELSE
			CONCAT2(ADR(str), ADR(arrayEnd2), ADR(str), SIZEOF(str));
		END_IF
		
	END_FOR
	
	CONCAT2(ADR(sPayloadPub), ADR(str), ADR(sPayloadPub), SIZEOF(sPayloadPub));
	
	(* lead acceleration x string *)
	str	:= ',"ax_lead":[';
	FOR i:=1 TO Get_IMU.Data_Length BY 1 DO
		CONCAT2(ADR(str), ADR(Get_IMU.AccX_Lead[i]), ADR(str), SIZEOF(str)); 
		
		IF i <> Get_IMU.Data_Length THEN
			CONCAT2(ADR(str), ADR(comma), ADR(str), SIZEOF(str));
		ELSE
			CONCAT2(ADR(str), ADR(arrayEnd2), ADR(str), SIZEOF(str));
		END_IF
		
	END_FOR
	
	CONCAT2(ADR(sPayloadPub), ADR(str), ADR(sPayloadPub), SIZEOF(sPayloadPub));
	
	(* lead acceleration y string *)
	str	:= ',"ay_lead":[';
	FOR i:=1 TO Get_IMU.Data_Length BY 1 DO
		CONCAT2(ADR(str), ADR(Get_IMU.AccY_Lead[i]), ADR(str), SIZEOF(str)); 
		
		IF i <> Get_IMU.Data_Length THEN
			CONCAT2(ADR(str), ADR(comma), ADR(str), SIZEOF(str));
		ELSE
			CONCAT2(ADR(str), ADR(arrayEnd2), ADR(str), SIZEOF(str));
		END_IF
		
	END_FOR
	
	CONCAT2(ADR(sPayloadPub), ADR(str), ADR(sPayloadPub), SIZEOF(sPayloadPub));
	
	(* lead acceleration z string *)
	str	:= ',"az_lead":[';
	FOR i:=1 TO Get_IMU.Data_Length BY 1 DO
		CONCAT2(ADR(str), ADR(Get_IMU.AccZ_Lead[i]), ADR(str), SIZEOF(str)); 
		
		IF i <> Get_IMU.Data_Length THEN
			CONCAT2(ADR(str), ADR(comma), ADR(str), SIZEOF(str));
		ELSE
			CONCAT2(ADR(str), ADR(arrayEnd2), ADR(str), SIZEOF(str));
		END_IF
		
	END_FOR
	
	CONCAT2(ADR(sPayloadPub), ADR(str), ADR(sPayloadPub), SIZEOF(sPayloadPub));
	
	(* lead pitch string *)
	str	:= ',"pitch_rear":[';
	FOR i:=1 TO Get_IMU.Data_Length BY 1 DO
		CONCAT2(ADR(str), ADR(Get_IMU.Pitch_Rear[i]), ADR(str), SIZEOF(str)); 
		
		IF i <> Get_IMU.Data_Length THEN
			CONCAT2(ADR(str), ADR(comma), ADR(str), SIZEOF(str));
		ELSE
			CONCAT2(ADR(str), ADR(arrayEnd2), ADR(str), SIZEOF(str));
		END_IF
		
	END_FOR
	
	CONCAT2(ADR(sPayloadPub), ADR(str), ADR(sPayloadPub), SIZEOF(sPayloadPub));
	
	(* rear roll string *)
	str	:= ',"roll_rear":[';
	FOR i:=1 TO Get_IMU.Data_Length BY 1 DO
		CONCAT2(ADR(str), ADR(Get_IMU.Roll_Rear[i]), ADR(str), SIZEOF(str)); 
		
		IF i <> Get_IMU.Data_Length THEN
			CONCAT2(ADR(str), ADR(comma), ADR(str), SIZEOF(str));
		ELSE
			CONCAT2(ADR(str), ADR(arrayEnd2), ADR(str), SIZEOF(str));
		END_IF
		
	END_FOR
	
	CONCAT2(ADR(sPayloadPub), ADR(str), ADR(sPayloadPub), SIZEOF(sPayloadPub));
	
	(* rear acceleration x string *)
	str	:= ',"ax_rear":[';
	FOR i:=1 TO Get_IMU.Data_Length BY 1 DO
		CONCAT2(ADR(str), ADR(Get_IMU.AccX_Rear[i]), ADR(str), SIZEOF(str)); 
		
		IF i <> Get_IMU.Data_Length THEN
			CONCAT2(ADR(str), ADR(comma), ADR(str), SIZEOF(str));
		ELSE
			CONCAT2(ADR(str), ADR(arrayEnd2), ADR(str), SIZEOF(str));
		END_IF
		
	END_FOR
	
	CONCAT2(ADR(sPayloadPub), ADR(str), ADR(sPayloadPub), SIZEOF(sPayloadPub));
	
	(* rear acceleration y string *)
	str	:= ',"ay_rear":[';
	FOR i:=1 TO Get_IMU.Data_Length BY 1 DO
		CONCAT2(ADR(str), ADR(Get_IMU.AccY_Rear[i]), ADR(str), SIZEOF(str)); 
		
		IF i <> Get_IMU.Data_Length THEN
			CONCAT2(ADR(str), ADR(comma), ADR(str), SIZEOF(str));
		ELSE
			CONCAT2(ADR(str), ADR(arrayEnd2), ADR(str), SIZEOF(str));
		END_IF
		
	END_FOR
	
	CONCAT2(ADR(sPayloadPub), ADR(str), ADR(sPayloadPub), SIZEOF(sPayloadPub));
	
	(* rear acceleration z string *)
	str	:= ',"az_rear":[';
	FOR i:=1 TO Get_IMU.Data_Length BY 1 DO
		CONCAT2(ADR(str), ADR(Get_IMU.AccZ_Rear[i]), ADR(str), SIZEOF(str)); 
		
		IF i <> Get_IMU.Data_Length THEN
			CONCAT2(ADR(str), ADR(comma), ADR(str), SIZEOF(str));
		ELSE
			CONCAT2(ADR(str), ADR(arrayEnd2), ADR(str), SIZEOF(str));
		END_IF
		
	END_FOR
	
	CONCAT2(ADR(sPayloadPub), ADR(str), ADR(sPayloadPub), SIZEOF(sPayloadPub));
	
	CONCAT2(ADR(sPayloadPub), ADR(msgEnd), ADR(sPayloadPub), SIZEOF(sPayloadPub)); //message ending
	
	(* publish message to subscribed topic *)
	IF Publish := fbMqttClient.Publish(sTopic:= sTopicPub, pPayload:= ADR(sPayloadPub), nPayloadSize:= LEN2(ADR(sPayloadPub)), eQoS:= TcIotMqttQos.AtMostOnceDelivery, bRetain:= FALSE, bQueue:= FALSE) THEN
		IF fbMqttClient.bError THEN
			// add your error logging here			
			hrErrorOccurred := fbMqttClient.hrErrorCode;
		ELSE
			Published 	:= TRUE;
		END_IF
		
	END_IF
	
END_IF

END_PROGRAM
